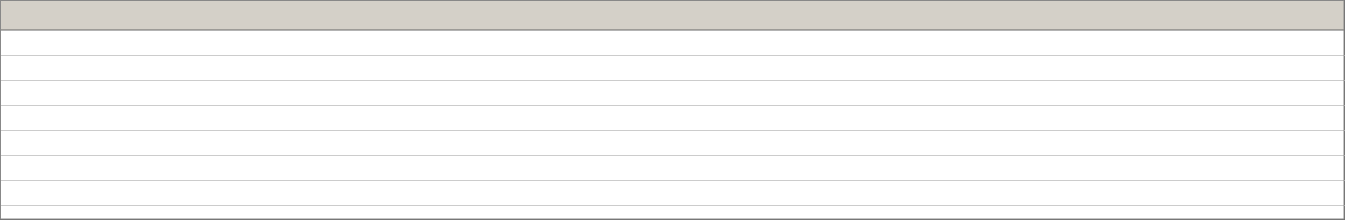
VISUALIZATION VISU_EV_EXTRAIT  // 1345x220
    Table (0,0 1345x220), data array: PRG_DEF_MANAGEMENT.EVENT_LIST
        p2232123230: PRG_DEF_MANAGEMENT.EVENT_LIST[INDEX].STATE_dt
        p511219082: PRG_DEF_MANAGEMENT.EVENT_LIST[INDEX].STATE_App
        p1755163831: PRG_DEF_MANAGEMENT.EVENT_LIST[INDEX].STATE_Path
        p4092479075: PRG_DEF_MANAGEMENT.EVENT_LIST[INDEX].STATE_Title
END_VISUALIZATION

(* stored: Version 1.1.0.1, ProductVersion 3.1.4024.10
   Visu VISU_EV_EXTRAIT: Id {bf005ee7-d279-44e6-9449-824b06a2755b} *)
